(* This function implements the Basic functions for the VAT590 needle valve*)
FUNCTION_BLOCK FB_VCN_VAT590 EXTENDS FB_Valve
VAR_INPUT
	bExtIlkOK	:	BOOL; //External Interlock, SET to TRUE if not used
//	fReqPos		:	REAL; //Requested position
//	bPurge		: 	BOOL := FALSE; // When purge is set the maximum threshold is ignored, has to be set evey cycle.
END_VAR
VAR_OUTPUT
	{attribute 'pytmc' := '
    pv:
	'}
	stVcnVat590	:	ST_VCN_VAT590; //Needle valve VAT590 structure
END_VAR
VAR CONSTANT
	cOpenPosition	:	REAL := 100000.0;   // Default position upper scale value
	cClosePosition	:	REAL := 0.0;        // Default position lower scale value
	cMaxPressure	:	REAL := 1000000.0;   // Default pressure upper scale value
	cLowPressure	:	REAL := 0;        // Default pressure lower scale value
END_VAR
VAR
	fCalcPosition : REAL := 0;
	fCalcPressure : REAL := 0;
	//eValveMode : E_VCN_VAT590;
	eValveModeSP : E_ControlModeSP;
	ePressureSens : E_PressureSensor;
	//eRemoteControl : E_AccessMode;
	eRemoteStatus : E_AccessMode;
	fReqPosition : REAL;
	fReqPressure : REAL;
	//bZero : BOOL;
	//bZeroDisabled : BOOL;
	bRemoteAccess : BOOL;
	//timer for zero function 
	tZeroDelay : TON := (PT := T#1S);
	//used for logging
	ePreviousState : E_VCN_VAT590;
 
	(*VAT590 Ethercat IO Interface*)
	//Ethercat Inputs
	i_nRawPosition       AT %I* : DINT;
	i_nRawPressure       AT %I* : DINT;
	i_eControlMode       AT %I* : E_ControlMode;
	i_eFatalError        AT %I* : E_FatalErrors;
	i_stGenStatus        AT %I* : ST_GeneralStatuses;
	i_stGenWarnings      AT %I* : ST_GeneralWarning;
	i_stExtnWarnings     AT %I* : ST_ExtendedWarning;
	//Ethercat outputs
	o_nRawPositionSP     AT %Q* : DINT;
	o_nRawPressureSP     AT %Q* : DINT;
	o_eCtrlModeSP        AT %Q* : E_ControlModeSP;
	o_stGenCtrlSP        AT %Q* : ST_GeneralControlSP;
END_VAR
VAR PERSISTENT
    fUpperLimit	: REAL;
END_VAR

(* Needle valve control FB
J. Govednik 2021-11-22

This FB should be used as a low level control block.

It provides:
Valve position ceiling
Interlock
Scaling

It could be used for:
Valve position/flow linearization
*)
ReadFromInput();

(*Checking which Control mode is selected*)
IF bExtIlkOK THEN
	CASE stVcnVat590.eValveControl OF
		E_VCN_VAT590.OpenValve:
			eValveModeSP := E_ControlModeSP.OpenValve;
		E_VCN_VAT590.CloseValve:
			eValveModeSP := E_ControlModeSP.CloseValve;
		E_VCN_VAT590.ManualControl:
			eValveModeSP := E_ControlModeSP.ManualControl;
			fReqPosition := LIMIT(0, stVcnVat590.fReqPosition, fUpperLimit);
		E_VCN_VAT590.PressureControl:
			eValveModeSP := E_ControlModeSP.PressureControl;
		E_VCN_VAT590.HoldValve:
			IF stVcnVat590.eControlMode = E_ControlMode.ManualControl OR
				stVcnVat590.eControlMode = E_ControlMode.PressureControl THEN
				eValveModeSP := E_ControlModeSP.HoldValve;
			END_IF
	END_CASE
ELSE
	fReqPosition := 0;
	eValveModeSP := E_ControlModeSP.CloseValve;
	stVcnVat590.eValveControl := E_VCN_VAT590.CloseValve;
END_IF

// Requested Position calculation
fCalcPosition := fReqPosition * (cOpenPosition-cClosePosition)/100 + cClosePosition;
fCalcPosition := LIMIT(cClosePosition, fCalcPosition, cOpenPosition); //The requested position SP should remain within this range

// Requested Pressure calculation
IF stVcnVat590.eValveControl = E_VCN_VAT590.PressureControl THEN
	CASE stVcnVat590.ePressureSensor OF
		E_PressureSensor.NOT_DEFINED:
			;
		E_PressureSensor.MKS500:
			;
	END_CASE
END_IF

fCalcPressure := fReqPressure * (cMaxPressure-cLowPressure)/100 + cLowPressure;
fCalcPressure := LIMIT(cLowPressure, fCalcPressure, cMaxPressure); //The requested pressure SP should remain within this range

//Zero function
IF stVcnVat590.stExtWarnings.ZeroDisabled OR tZeroDelay.Q THEN
	stVcnVat590.bZero := FALSE;
END_IF
tZeroDelay.IN := stVcnVat590.bZero;
tZeroDelay();

//Set Remote Access
IF eRemoteStatus <> stVcnVat590.eRemoteControl THEN
	//bRemoteAccess := NOT bRemoteAccess;
	bRemoteAccess := FALSE; //Don't switch remote control for now
END_IF

(*Soft IO Mapping*)
WriteToOutput();

(*Load or save the persistent variables*)
ACT_Persistent();


(*
	IF stVcnVat590.eValveControl = E_VCN_VAT590.OpenValve THEN
		stVcnVat590.fReqPosition := stVcnVat590.fUpperLimit;(*Percentage*)
	ELSIF stVcnVat590.eValveControl = E_VCN_VAT590.CloseValve THEN
		stVcnVat590.fReqPosition := 0; (*Percentage*)
	ELSIF (stVcnVat590.eValveControl = E_VCN_VAT590.ManualControl) (*AND (iq_stVCN.xOPN_SW)*) THEN
		;
	ELSIF stVcnVat590.eValveControl = E_VCN_VAT590.PressureControl THEN
		IF (bPurge) THEN
			stVcnVat590.fReqPosition := LIMIT(0, fReqPos, 100); 
		ELSE 
			stVcnVat590.fReqPosition := LIMIT(0, fReqPos, stVcnVat590.fUpperLimit); 
		END_IF
	END_IF
*)

ACTION ACT_Logger:
// ILK logger

IF NOT (stVcnVat590.bIlkOK ) AND NOT(ePreviousState = E_VCN_VAT590.CloseValve) THEN
 		fbLogger(sMsg:='Lost interlock ok bit while valve was open.', eSevr:=TcEventSeverity.Critical);  	
END_IF


//Control STATE Logger  
IF ePreviousState <> stVcnVat590.eValveControl THEN
	  CASE stVcnVat590.eValveControl OF
		E_VCN_VAT590.ManualControl:
			fbLogger(sMsg:='Valve in manual control mode', eSevr:=TcEventSeverity.Warning);
		E_VCN_VAT590.HoldValve:
			fbLogger(sMsg:='Valve in hold control mode', eSevr:=TcEventSeverity.Warning);
		E_VCN_VAT590.OpenValve:
			fbLogger(sMsg:='Valve Open.', eSevr:=TcEventSeverity.Info);
		E_VCN_VAT590.PressureControl:
			fbLogger(sMsg:='Valve in pressure control mode.', eSevr:=TcEventSeverity.Info);
		E_VCN_VAT590.CloseValve:
			fbLogger(sMsg:='Valve closed.', eSevr:=TcEventSeverity.Info);
	  END_CASE
	  ePreviousState := stVcnVat590.eValveControl;  
  END_IF
 

// Log valve open
tAction(CLK:= (stVcnVat590.eValveControl = E_VCN_VAT590.OpenValve) );
IF tAction.Q THEN fbLogger(sMsg:='Valve commanded to fully open', eSevr:=TcEventSeverity.Info); END_IF
END_ACTION

ACTION ACT_Persistent:
(*On first PLC pass, load the persistent value into the structrue variable*)
IF (bRestorePersistentData) THEN
	bRestorePersistentData	:= FALSE;
	IF (fUpperLimit <> 0) THEN
		stVcnVat590.fUpperLimit := fUpperLimit;
	END_IF;
	
END_IF
(*Check if a new value has been written in the structure variable copy it to the persistent variable*)
IF NOT (stVcnVat590.fUpperLimit = fUpperLimit) THEN
	fUpperLimit := stVcnVat590.fUpperLimit;
	//fbWritePersistentData(NETID:='', PORT:=851, START:=TRUE, TMOUT:=T#1s );
ELSE
     // fbWritePersistentData( START:=FALSE);
END_IF;
END_ACTION

METHOD M_SetThrottle : BOOL
VAR_INPUT
	rUpperLimit	:	REAL;
END_VAR

stVcnVat590.fUpperLimit := LIMIT(0, rUpperLimit, 100);
END_METHOD

METHOD M_ValveControl : BOOL
VAR_INPUT
	state : E_VCN_VAT590; // Set Control modes
END_VAR
stVcnVat590.eValveControl := state;
END_METHOD

ACTION ReadFromInput:
//Read from EPICS
fUpperLimit := LIMIT(0, stVcnVat590.fUpperLimit, 100);
fReqPosition := LIMIT(0, stVcnVat590.fReqPosition, 100);
fReqPressure := stVcnVat590.fReqPressure;

//Read from VAT valve
stVcnVat590.eControlMode := i_eControlMode;
stVcnVat590.eFatalErrors := i_eFatalError;
stVcnVat590.nRawPosition := i_nRawPosition;
stVcnVat590.nRawPressure := i_nRawPressure;
//Mapping General statuses
stVcnVat590.stGenStatus.FieldBusDatavalid := i_stGenStatus.Bit0FieldBusDatavalid;
stVcnVat590.stGenStatus.ZeroExecuted := i_stGenStatus.Bit1ZeroExecuted;
stVcnVat590.stGenStatus.PingPongRxBit := i_stGenStatus.Bit2PingPongRxBit;
stVcnVat590.stGenStatus.PressureSimulation := i_stGenStatus.Bit3PressureSimulation;
stVcnVat590.stGenStatus.PressureSPReached := i_stGenStatus.Bit4PressureSPReached;
stVcnVat590.stGenStatus.WarningsActive := i_stGenStatus.Bit9WarningsActive;
//Mapping General warnings
stVcnVat590.stGenWarnings.ServiceRequest := i_stGenWarnings.Bit0ServiceRequest;
stVcnVat590.stGenWarnings.PowerFailureBattery := i_stGenWarnings.Bit3PowerFailureBattery;
stVcnVat590.stGenWarnings.SensMeasUnitFault := i_stGenWarnings.Bit10SensMeasUnitFault;
//Mapping Extended warnings
stVcnVat590.stExtWarnings.RemoteControlNotPossible := i_stExtnWarnings.Bit0RemoteControlNotPossible;
stVcnVat590.stExtWarnings.ControlModeSPNotAllowed := i_stExtnWarnings.Bit1ControlModeSPNotAllowed;
stVcnVat590.stExtWarnings.ZeroDisabled := i_stExtnWarnings.Bit2ZeroDisabled;
stVcnVat590.stExtWarnings.PFODeactivated := i_stExtnWarnings.Bit3PFODeactivated;
stVcnVat590.stExtWarnings.PressureSPOutOfRange := i_stExtnWarnings.Bit5PressureSPOutOfRange;
stVcnVat590.stExtWarnings.PositionSPOutOfRange := i_stExtnWarnings.Bit6PositionSPOutOfRange;
stVcnVat590.stExtWarnings.CtrlSPOutOfRange := i_stExtnWarnings.Bit10CtrlSPOutOfRange;
stVcnVat590.stExtWarnings.GeneralCtrlSPOutOfRange := i_stExtnWarnings.Bit11GeneralCtrlSPOutOfRange;
stVcnVat590.stExtWarnings.ProcDataSettingsNotvalid := i_stExtnWarnings.Bit12ProcDataSettingsNotvalid;
//Read Remote status 
eRemoteStatus.0 := i_stGenStatus.Bit7AccessModeBit0;
eRemoteStatus.1 := i_stGenStatus.Bit8AccessModeBit1;
END_ACTION

ACTION WriteToOutput:
//Write to EPICS
stVcnVat590.bIlkOK := bExtIlkOK;
stVcnVat590.nPositionSP := REAL_TO_DINT(fCalcPosition);
stVcnVat590.nPressureSP := REAL_TO_DINT(fCalcPressure);
stVcnVat590.eRemoteControl := eRemoteStatus;
stVcnVat590.fReqPosition := fReqPosition;
stVcnVat590.fReqPressure := fReqPressure;

//Write to VAT valve
o_eCtrlModeSP := eValveModeSP;
o_nRawPositionSP := REAL_TO_DINT(fCalcPosition);
o_nRawPressureSP := REAL_TO_DINT(fCalcPressure);
o_stGenCtrlSP.Bit0ExecuteZero := stVcnVat590.bZero;
o_stGenCtrlSP.Bit4AccessMode := bRemoteAccess;
END_ACTION

END_FUNCTION_BLOCK

(* stored: Version 1.1.0.1, ProductVersion 3.1.4022.18
   POU FB_VCN_VAT590: Id {4758ecab-cc0c-4c37-8981-9d3a1c0c082a}, SpecialFunc None
   Action ACT_Logger: Id {e05977be-b3df-4692-b1e1-f426b01665a8}
   Action ACT_Persistent: Id {e5168615-6ef3-4946-b318-5dac9816d744}
   Method M_SetThrottle: Id {bc87ba94-efcb-4d7b-ace0-cb07482f478f}
   Method M_ValveControl: Id {25066385-eb5f-47fb-8ac4-a5fcdc50740f}
   Action ReadFromInput: Id {2b46db7d-12fe-424a-afdf-e2d60ed01bdb}
   Action WriteToOutput: Id {d6e20cf1-2c45-411b-b669-d1005d8dcb97} *)
